# EPICS autosave request: iocBoot/iocelveFlowESmobile/auto_settings.req
file "elveFlowESmobile.req",
